(* IEC 61131-3 sources: eCockpitGit/test_project/src/%F%00 Library/%F%Common Functions/%F%Dynamic Array/%F%Dynamic Sorted Array Helpers, 2 files *)

(* ---- %POU%FU_wDynamicSortedArrayFromStruct.st ---- *)
FUNCTION FU_wDynamicSortedArrayFromStruct : SLMResult
VAR_INPUT
	dynArr				:REFERENCE TO FB_wDynamicSortedArray;
	reader				:ITF_StructReaderBase;
END_VAR
VAR
	length				:WORD;
	i					:WORD;
END_VAR
(*%!%__DELIMITER__%!%*)
IF reader.valueType = EStructType.tArray THEN
	dynArr.empty();
	reader.enterObjectArray();
	length												:=		reader.amountInSelection;
	FU_wDynamicSortedArrayFromStruct					:=		dynArr.allocate(size:=length);
	IF FU_wDynamicSortedArrayFromStruct.success AND length > 0 THEN
		FOR i := 1 TO length DO
			IF reader.nextArray() <> EStructType.none THEN
				FU_wDynamicSortedArrayFromStruct		:=		dynArr.addElement(element:=reader.readWord());
				IF NOT(FU_wDynamicSortedArrayFromStruct.success) THEN
					EXIT;
				END_IF
			ELSE
				EXIT;
			END_IF
		END_FOR
	END_IF
	reader.exitObjectArray();
END_IF

(* ---- %POU%FU_wDynamicSortedArrayToStruct.st ---- *)
FUNCTION FU_wDynamicSortedArrayToStruct : SLMResult
VAR_INPUT
	dynArr				:REFERENCE TO FB_wDynamicSortedArray;
	writer				:ITF_StructWriterBase;
END_VAR
VAR
	i					:WORD;
	buffer				:WORD;
END_VAR
(*%!%__DELIMITER__%!%*)
writer.arrayStart(singleLine:=TRUE);
IF dynArr.S_lenght > 0 THEN
	FOR i := 0 TO dynArr.S_lenght - 1 DO
		dynArr.getElementByIndex(index:=i,element=>buffer);
		writer.writeDint(value:=buffer);
	END_FOR
END_IF
writer.structEnd();
